/// Event structure
TYPE ST_Event EXTENDS ST_EventBase:
STRUCT
	dtRaiseTime			: DT;
	dtQuitTime			: DT;	
END_STRUCT
END_TYPE

(* stored: Version 1.1.0.1
   DUT ST_Event: Id {ff39c85d-5c87-4bc5-84de-330d6e07205e} *)
